// TIA Portal V16 export
// export: Created 2024-12-03T15:41:45.8331022Z, ExportSetting WithReadOnly, DisplayName Totally Integrated Automation Portal, DisplayVersion V16 Update 6, DisplayName TIA Portal Version Control Interface, DisplayVersion V16 Update 2, DisplayName TIA Portal Openness, DisplayVersion V16 Update 6, DisplayName TIA Portal Teamcenter Gateway, DisplayVersion V16, DisplayName SINAMICS Startdrive Advanced, DisplayVersion V16 Update 5, DisplayName SINAMICS Startdrive G130, G150, S120, S150, SINAMICS MV, S210, DisplayVersion V16 Update 5, DisplayName SINAMICS Startdrive G110M, G120, G120C, G120D, G120P, G115D, DisplayVersion V16 Update 5, DisplayName STEP 7 Professional, DisplayVersion V16 Update 6, DisplayName STEP 7 Safety, DisplayVersion V16, DisplayName WinCC Advanced / Unified PC, DisplayVersion V16 Update 6
TYPE "Nord_Drive_SK5xx_Out_Data_UDT"
// stored: CreationDate 2024-12-03T06:55:59.9692037Z, InterfaceModifiedDate 2023-12-19T13:50:46.8800733Z, IsConsistent true, LibraryConformanceStatus The object is library-conformant., ModifiedDate 2023-12-19T13:50:46.8800733Z
   STRUCT
      xStart48011_Takt : Bool;   // See P480
      xStart48012_Home : Bool;   // See P480
      xCrtlData : Bool;   // 1 = Valid process data
      CmdRightDirection : Bool;   // Cmd turning right
      CmdLeftDirection : Bool;   // Cmd turning left
      Reserve_1 : Bool;   // Reserved
      Parameterset_LSB : Bool;   // 0 = Par set 1 / 1 = Par set 2 / 2 = Par set 3 / 3 = Par set 4
      Parameterset_MSB : Bool;   // 0 = Par set 1 / 1 = Par set 2 / 2 = Par set 3 / 3 = Par set 4
      CmdReadyForOPeration : Bool;   // 1 = Ready for operation
      ActivatePower : Bool;   // 0 = Cut off voltage
      EmergencyOk : Bool;   // 0 = Activeer noodstop
      EnableOperation : Bool;   // 1 = Enable operation
      EnableRampGenerator : Bool;   // 1 = Enable ramp generator
      EnableSetPointRampGenerator : Bool;   // 1 = Setpoint on ramp generator enabled
      xEnSetp : Bool;   // 1 = Selected ramp generator setpoint is activated
      ResetError : Bool;   // FP = Acknowkedge all errors
      MotorSetpointSpeed : Int;   // Motor speed set point
      DigitalOutputs : Struct   // Digital outputs
         spare_7 : Byte;
         Relay_1 : Bool;   // Relay output 1
         Relay_2 : Bool;   // Relay output 2
         Output_1 : Bool;   // Digital Output 1 (SK550 only)
         Output_2 : Bool;   // Digital Output 2 (SK550 only)
         spare_3 : Bool;
         spare_4 : Bool;
         spare_5 : Bool;
         spare_6 : Bool;
      END_STRUCT;
      Reserve_2 : Int := 0;   // Reserve
   END_STRUCT;
END_TYPE
